// TIA Portal V20 export
TYPE "LER_typeThicknessTrackingData"
// stored: Access Published
   STRUCT
      finished { ExternalWritable := 'False'} : Bool;
      result { ExternalWritable := 'False'} : Bool;
      data { ExternalWritable := 'False'} : Array[0..3] of Real;
   END_STRUCT;
END_TYPE
